FUNCTION_BLOCK Skill_LoadDeliverReturn EXTENDS FB_2_Template_Skill
VAR_INPUT
	Rob: POINTER TO FB_2_ROB_AMR;
	sPickReference: STRING;
END_VAR
VAR_OUTPUT
	
END_VAR
VAR
	
	ActiveBAFinished: BOOL;
	ccc: BOOL;
END_VAR

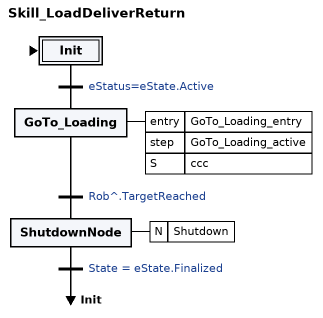
INITIAL_STEP Init:
END_STEP
TRANSITION FROM Init TO GoTo_Loading
    := eStatus=eState.Active;
END_TRANSITION
STEP GoTo_Loading:
    GoTo_Loading_entry(P1);  // entry action
    GoTo_Loading_active(N);  // step action
    ccc(S);
END_STEP
TRANSITION FROM GoTo_Loading TO ShutdownNode
    := Rob^.TargetReached;
END_TRANSITION
STEP ShutdownNode:
    Shutdown(N);
END_STEP
TRANSITION FROM ShutdownNode TO Init
    := State = eState.Finalized;
END_TRANSITION

ACTION GoTo_Loading_active:

END_ACTION

ACTION GoTo_Loading_entry:
Rob^.NavigateToGoal(goal := 'Station1');
END_ACTION

END_FUNCTION_BLOCK

(* stored: Version 1.1.0.1, ProductVersion 3.1.4026.18
   POU Skill_LoadDeliverReturn: Id {8977347b-02ee-433d-9081-1576e654bc94}, SpecialFunc None
   Action GoTo_Loading_active: Id {64c92707-b03c-4a2e-9acb-24760aeeb714}
   Action GoTo_Loading_entry: Id {ac9dceb2-bfc1-45d4-b847-bffce732acdb} *)
